{attribute 'qualified_only'}
VAR_GLOBAL
END_VAR

(* stored: Version 1.1.0.1, ProductVersion 3.1.4024.6
   GVL GVL_1: Id {f84502fe-dc42-4a31-a311-32c9b80be47b} *)
